FUNCTION_BLOCK FB_AttFFO
VAR_IN_OUT
    stMotionStage: DUT_MotionStage;
    fbFFHWO: FB_HardwareFFOutput;
END_VAR
VAR_OUTPUT
    bIsNotMoving: BOOL;
END_VAR
VAR
    fbFF: FB_FastFault := (i_Desc := 'Device is moving',
                           i_TypeCode := 16#2100,
                           i_xAutoReset := TRUE);
END_VAR

bIsNotMoving := NOT stMotionStage.Axis.Status.Moving;
fbFF(i_DevName := stMotionStage.sName,
     i_xOK := bIsNotMoving,
     io_fbFFHWO := fbFFHWO);

END_FUNCTION_BLOCK

(* stored: Version 1.1.0.1, ProductVersion 3.1.4022.18
   POU FB_AttFFO: Id {8aee63dd-8a4c-007a-10c6-ebcc0e6cea6a}, SpecialFunc None *)
